Fanuc TP program (LS listing): SYSV_KEYP.LS

/PROG  SYSV_KEYP
/ATTR
OWNER		= MNEDITOR;
COMMENT		= "sysvar probe";
PROG_SIZE	= 0;
CREATE		= DATE 26-01-01  TIME 00:00:00;
MODIFIED	= DATE 26-01-01  TIME 00:00:00;
FILE_NAME	= ;
VERSION		= 0;
LINE_COUNT	= 4;
MEMORY_SIZE	= 0;
PROTECT		= READ_WRITE;
TCD:  STACK_SIZE	= 0,
      TASK_PRIORITY	= 50,
      TIME_SLICE	= 0,
      BUSY_LAMP_OFF	= 0,
      ABORT_REQUEST	= 0,
      PAUSE_REQUEST	= 0;
DEFAULT_GROUP	= 1,*,*,*,*;
CONTROL_CODE	= 00000000 00000000;
/MN
   1:  !sysvar probe ;
   2:  R[155]=0    ;
   3:  R[154]=$MSKKEY_PANL    ;
   4:  R[155]=1    ;
/POS
/END
